FUNCTION_BLOCK CM_DockingClamps EXTENDS CM_Base

VAR_INPUT
	i_stSettings : ST_SettingsDockingClamps;
END_VAR

VAR
	// Control Modules
	s_cmValveDockingClampsUpper : CM_ValveWithDoubleFB;
	s_cmValveDockingClampsLower : CM_ValveWithDoubleFB;
	
	// Request
	s_bReqOpen : BOOL;
	s_bReqClose : BOOL;
	
	// Status
	s_bStaIsOpened : BOOL; 
	s_bStaIsClosed : BOOL;
	
	{attribute: 'Hide'}
	s_bStaClamps : BOOL; //FALSE = Closed, TRUE = Opened
	
	// Alarms
	
	// Timers
END_VAR


SUPER^();

METHOD PROTECTED _m_Alarms : BOOL

IF NOT SUPER^._m_Alarms() THEN
	RETURN;
END_IF

s_bStaError := 
	s_cmValveDockingClampsUpper.p_bStaError
	OR s_cmValveDockingClampsLower.p_bStaError;

_m_Alarms := TRUE;
END_METHOD

METHOD PROTECTED _m_Devices : BOOL

IF NOT SUPER^._m_Devices() THEN
	RETURN;
END_IF

//Call lower-layer devices
s_cmValveDockingClampsUpper(
	i_bReqEnable	:= i_bReqEnable, 
	i_eCtrlMode		:= i_eCtrlMode,
	i_bCmdReset		:= i_bCmdReset,
	i_sCmName		:= 'Upper Docking Clamps'); 
	
s_cmValveDockingClampsLower(
	i_bReqEnable	:= i_bReqEnable, 
	i_eCtrlMode		:= i_eCtrlMode,
	i_bCmdReset		:= i_bCmdReset,
	i_sCmName		:= 'Lower Docking Clamps');

//Control lower-layer devcies
IF s_bReqOpen THEN
	s_cmValveDockingClampsUpper.m_Off();
	s_cmValveDockingClampsLower.m_Off();
ELSIF s_bReqClose THEN
	s_cmValveDockingClampsUpper.m_On();
	s_cmValveDockingClampsLower.m_On();
ELSE
	s_cmValveDockingClampsUpper.m_Stop();
	s_cmValveDockingClampsLower.m_Stop();
END_IF
	
//Statusses
s_bStaIsOpened := s_cmValveDockingClampsUpper.p_bStaIsOff AND s_cmValveDockingClampsLower.p_bStaIsOff;
s_bStaIsClosed := s_cmValveDockingClampsUpper.p_bStaIsOn AND s_cmValveDockingClampsLower.p_bStaIsOn;

s_bStaClamps := NOT(s_bStaIsOpened) AND s_bStaIsClosed; 

_m_Devices := TRUE;
END_METHOD

METHOD PROTECTED _m_Hmi : BOOL

IF NOT SUPER^._m_Hmi() THEN
	RETURN;
END_IF

_m_Hmi := TRUE;
END_METHOD

METHOD PROTECTED _m_Init : BOOL
IF NOT SUPER^._m_Init() THEN
	RETURN;
END_IF

s_cmValveDockingClampsUpper.i_stSettings.tValveOffTimeout := i_stSettings.tClampsOpenTimeout;
s_cmValveDockingClampsUpper.i_stSettings.tValveOnTimeout := i_stSettings.tClampsCloseTimeout;

s_cmValveDockingClampsLower.i_stSettings.tValveOffTimeout := i_stSettings.tClampsOpenTimeout;
s_cmValveDockingClampsLower.i_stSettings.tValveOnTimeout := i_stSettings.tClampsCloseTimeout;

_m_Init := TRUE;
END_METHOD

METHOD PROTECTED _m_Inputs : BOOL

IF NOT SUPER^._m_Inputs() THEN
	RETURN;
END_IF

_m_Inputs := TRUE;
END_METHOD

METHOD PROTECTED _m_Outputs : BOOL

IF NOT SUPER^._m_Outputs() THEN
	RETURN;
END_IF

_m_Outputs := TRUE;
END_METHOD

METHOD PUBLIC m_Close : BOOL

IF NOT i_bReqEnable THEN 
	RETURN;
END_IF

s_bReqOpen := FALSE;
s_bReqClose := TRUE;

m_Close := TRUE;
END_METHOD

METHOD PUBLIC m_Open : BOOL

IF NOT i_bReqEnable THEN 
	RETURN;
END_IF

s_bReqOpen := TRUE;
s_bReqClose := FALSE;

m_Open := TRUE;
END_METHOD

METHOD PUBLIC m_Stop : BOOL

IF NOT i_bReqEnable THEN 
	RETURN;
END_IF

s_bReqOpen := FALSE;
s_bReqClose := FALSE;

m_Stop := TRUE;
END_METHOD

{attribute 'monitoring':='call'}
PROPERTY PUBLIC p_bStaClamps : BOOL
GET

p_bStaClamps := s_bStaClamps;
END_GET
END_PROPERTY

{attribute 'monitoring':='call'}
PROPERTY PUBLIC p_bStaIsClosed : BOOL
GET

p_bStaIsClosed := s_bStaIsOpened;
END_GET
END_PROPERTY

{attribute 'monitoring':='call'}
PROPERTY PUBLIC p_bStaIsOpened : BOOL
GET

p_bStaIsOpened := s_bStaIsClosed;
END_GET
END_PROPERTY

END_FUNCTION_BLOCK

(* stored: Version 1.1.0.1, ProductVersion 3.1.4024.12
   POU CM_DockingClamps: Id {707e5e9b-ec6e-4cfc-802c-8528e1988b9b}, SpecialFunc None
   Folder Methods: Id {ffeb2278-57ae-456a-853a-75bd02373c15}
   Folder Properties: Id {4d103486-2a68-4a14-b19c-bb4ac96a75be}
   Method _m_Alarms: Id {f33d2966-4692-4c6e-951b-66a70933eb5b}
   Method _m_Devices: Id {bda56788-e543-4c1d-a9c1-3bcca55e5a0e}
   Method _m_Hmi: Id {161a2353-3fa8-4a12-bcb9-7cd8e64b8355}
   Method _m_Init: Id {246b5534-eba6-48a2-9d8e-ab08715419e1}
   Method _m_Inputs: Id {b00b0ad1-683f-43da-8632-a01c1971348b}
   Method _m_Outputs: Id {2d786b78-4b0b-41c0-9cad-0cfe793a91e3}
   Method m_Close: Id {f0019df8-b38e-4360-b666-0a6461ce5434}
   Method m_Open: Id {ee548796-f12d-4452-8126-b68ccf293d10}
   Method m_Stop: Id {baaf2f36-9288-4025-b2f3-7b96489fad9e}
   Property p_bStaClamps: Id {59914008-3706-4d6d-a885-02d051be215d}
   Get Get: Id {28aeb0a5-88dd-402f-b72e-702c29341244}
   Property p_bStaIsClosed: Id {b5985041-12b2-4457-a7ba-6467f6192394}
   Get Get: Id {9f3c5d38-a6b3-4848-a2c8-7bb49acc32d4}
   Property p_bStaIsOpened: Id {1f74d561-75ba-4c24-9a4d-2d3cc0be044a}
   Get Get: Id {096de774-de50-4249-bc2b-268c7b612ac8} *)
